Omron Sysmac Studio project Benim_Fonk (Sysmac Studio 1.65.0.64007, StandardProject)

# Controller new_Controller_0: NX1P2-1040DT1 version 1.69
Task PrimaryTask (priority 4, period or condition 2000): Program0

VAR_GLOBAL
    AI_Value2 : REAL;
    OnOff : BOOL;
END_VAR

PROGRAM Program1
VAR
    EnableIn : BOOL;
    EnableOut : BOOL;
    Filtreleme_Start : BOOL;
    Pulse : BOOL;
    Pulse_prev : BOOL;
    Pulse_edge : BOOL;
    Sayici : INT;
    AnalogInput : REAL;
    AnalogArry : ARRAY[1..5] OF REAL;
    Sayici_prev : INT;
    Sayici_chg : BOOL;
    InitDone : BOOL;
    AverageValue : REAL;
END_VAR
(* 
   RUNG 0
   EnableIn -> EnableOut
*)
EnableOut := EnableIn;


(* 
   RUNG 1
   Pulse YÜKSELENKENAR-edge yakala ve Sayici artır
   (Filtreleme_Start TRUE iken)
*)
Pulse_edge := Pulse AND NOT Pulse_prev;
Pulse_prev := Pulse;

IF Filtreleme_Start AND Pulse_edge THEN
    Sayici := Sayici + INT#1;
END_IF;


(* 
   RUNG 2–6 (Optimize)
   Sayici değiştiğinde (Up mantığı gibi tek sefer) ve 1..5 aralığındaysa
   AnalogArry[Sayici] := AnalogInput
 *)
IF NOT InitDone THEN
    Sayici_chg := FALSE;        (* ilk task'ta tetik üretme *)
    Sayici_prev := Sayici;      (* başlangıç referansı *)
    InitDone := TRUE;
ELSE
    Sayici_chg := (Sayici <> Sayici_prev);
    Sayici_prev := Sayici;
END_IF;

IF Sayici_chg AND (Sayici >= INT#1) AND (Sayici <= INT#5) THEN
    AnalogArry[Sayici] := AnalogInput;

    (* 
       RUNG 6 içindeki AryMean
 *)
    IF Sayici = INT#5 THEN
        AverageValue :=
            (AnalogArry[1] + AnalogArry[2] + AnalogArry[3] + AnalogArry[4] + AnalogArry[5]) / REAL#5.0;
    END_IF;
END_IF;


(* 
   RUNG 7
   Sayici > 5 olunca Sayici'yi 1'e çek
   (Ladder'da Up+MOVE var; burada wrap mantığıyla aynı sonucu verir)
 *)
IF Sayici > INT#5 THEN
    Sayici := INT#1;
END_IF;
END_PROGRAM

PROGRAM Program0
VAR
    Scale_Value : REAL;
    Scale_X0 : REAL;
    Scale_Y0 : REAL;
    Scale_X1 : REAL;
    Scale_Y1 : REAL;
    Scale_Out : REAL;
    Lim_Min : REAL;
    Lim_Max : REAL;
    Lim_Out : REAL;
    Analog_Input : REAL;
    InputMin : REAL;
    OutputMin : REAL;
    OutputMax : REAL;
    BasinsDeg : REAL;
    InputMax : REAL;
    BenimFiltre_5liOrt : Filtreleme;
    Ton_Pulse : TON;
    Pulse_200ms : BOOL;
    Ortalama_Deger : REAL;
    OnOff : BOOL;
END_VAR
VAR_EXTERNAL
    AI_Value2 : REAL;
END_VAR
VAR
    _t1 : BOOL;
    _p2 : BOOL;
END_VAR

(* Section Section0: ladder, written here as Structured Text *)

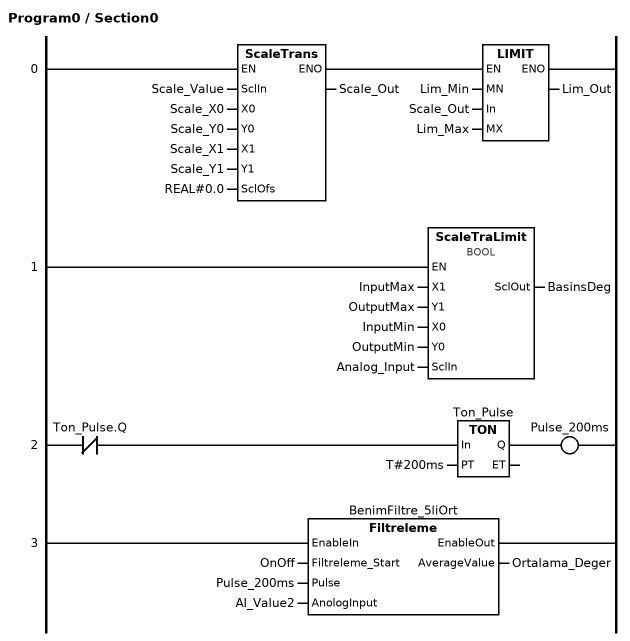
(* Rung 0 *)
Scale_Out := ScaleTrans(SclIn := Scale_Value, X0 := Scale_X0, Y0 := Scale_Y0, X1 := Scale_X1, Y1 := Scale_Y1, SclOfs := REAL#0.0);
Lim_Out := LIMIT(MN := Lim_Min, In := Scale_Out, MX := Lim_Max);
(* Rung 1 *)
_t1 := ScaleTraLimit(X1 := InputMax, Y1 := OutputMax, X0 := InputMin, Y0 := OutputMin, SclIn := Analog_Input, SclOut => BasinsDeg);
(* Rung 2 *)
_p2 := NOT Ton_Pulse.Q;
Ton_Pulse(In := _p2, PT := T#200ms);
Pulse_200ms := Ton_Pulse.Q;
(* Rung 3 *)
BenimFiltre_5liOrt(EnableIn := TRUE, Filtreleme_Start := OnOff, Pulse := Pulse_200ms, AnologInput := AI_Value2, AverageValue => Ortalama_Deger);
END_PROGRAM

FUNCTION ScaleTraLimit : BOOL
VAR
    Scl_Out_Temp : REAL;
END_VAR
VAR_INPUT
    X1 : REAL;
    Y1 : REAL;
    X0 : REAL;
    Y0 : REAL;
    SclIn : REAL;
END_VAR
VAR_OUTPUT
    SclOut : REAL;
END_VAR
(* ladder, written here as Structured Text *)

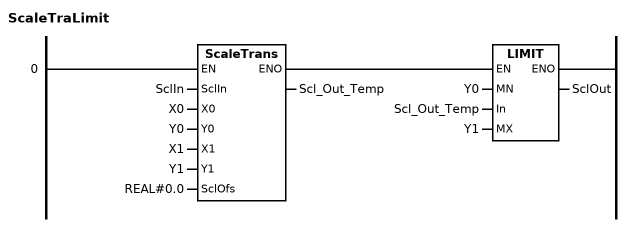
(* Rung 0 *)
Scl_Out_Temp := ScaleTrans(SclIn := SclIn, X0 := X0, Y0 := Y0, X1 := X1, Y1 := Y1, SclOfs := REAL#0.0);
SclOut := LIMIT(MN := Y0, In := Scl_Out_Temp, MX := Y1);
END_FUNCTION

FUNCTION Function0 : BOOL
VAR
    EnableIn : BOOL;
    EnableOut : BOOL;
    Filtreleme_Start : BOOL;
    Pulse : BOOL;
    Pulse_prev : BOOL;
    Pulse_edge : BOOL;
    Sayici : INT;
    AnalogInput : REAL;
    AnalogArry : ARRAY[1..5] OF REAL;
    Sayici_prev : INT;
    Sayici_chg : BOOL;
    InitDone : BOOL;
END_VAR
(* Rung 0 *)
EnableOut := EnableIn;

(* Rung 1 *)
Pulse_edge := Pulse AND NOT Pulse_prev;
Pulse_prev := Pulse;

IF Filtreleme_Start AND Pulse_edge THEN
    Sayici := Sayici + INT#1;
END_IF;

(* Rung 2–6 *)
IF NOT InitDone THEN
    Sayici_chg := FALSE;
    Sayici_prev := Sayici;
    InitDone := TRUE;
ELSE
    Sayici_chg := (Sayici <> Sayici_prev);
    Sayici_prev := Sayici;
END_IF;

IF Sayici_chg AND (Sayici >= INT#1) AND (Sayici <= INT#5) THEN
    AnalogArry[Sayici] := AnalogInput;
END_IF;
END_FUNCTION

FUNCTION_BLOCK Filtreleme
VAR
    Sayici : INT;
    AnologArry : ARRAY[1..5] OF REAL;
END_VAR
VAR_INPUT
    EnableIn : BOOL;
END_VAR
VAR_OUTPUT
    EnableOut : BOOL;
END_VAR
VAR_INPUT
    Filtreleme_Start : BOOL;
    Pulse : BOOL;
    AnologInput : REAL;
END_VAR
VAR_OUTPUT
    AverageValue : REAL;
END_VAR
VAR
    _e1 : R_TRIG;
    _e2 : R_TRIG;
    _e3 : R_TRIG;
    _e4 : R_TRIG;
    _e5 : R_TRIG;
    _e6 : R_TRIG;
    _e7 : R_TRIG;
END_VAR
(* ladder, written here as Structured Text *)

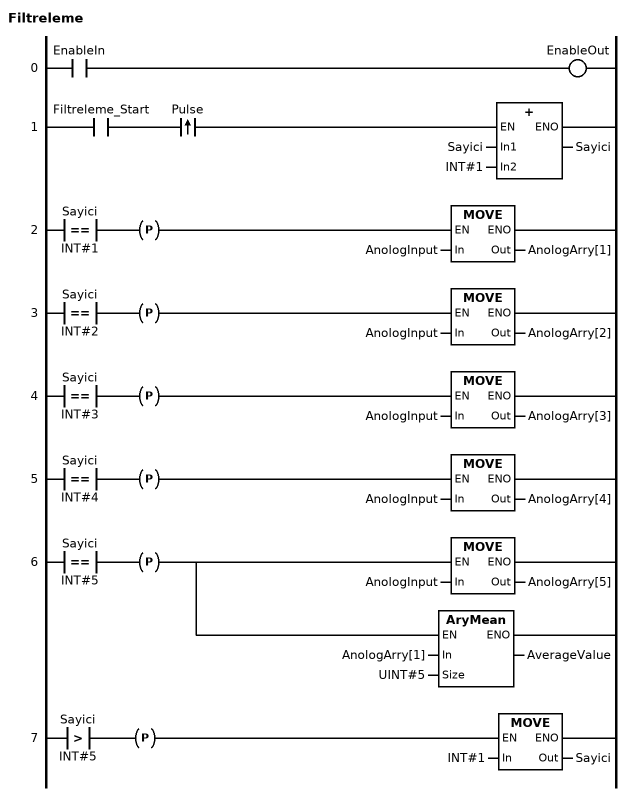
(* Rung 0 *)
EnableOut := EnableIn;
(* Rung 1 *)
_e1(CLK := Pulse);
IF Filtreleme_Start AND _e1.Q THEN Sayici := Sayici + INT#1; END_IF;
(* Rung 2 *)
_e2(CLK := Sayici = INT#1);
IF _e2.Q THEN AnologArry[1] := AnologInput; END_IF;
(* Rung 3 *)
_e3(CLK := Sayici = INT#2);
IF _e3.Q THEN AnologArry[2] := AnologInput; END_IF;
(* Rung 4 *)
_e4(CLK := Sayici = INT#3);
IF _e4.Q THEN AnologArry[3] := AnologInput; END_IF;
(* Rung 5 *)
_e5(CLK := Sayici = INT#4);
IF _e5.Q THEN AnologArry[4] := AnologInput; END_IF;
(* Rung 6 *)
_e6(CLK := Sayici = INT#5);
IF _e6.Q THEN
    AnologArry[5] := AnologInput;
    AverageValue := AryMean(In := AnologArry[1], Size := UINT#5);
END_IF;
(* Rung 7 *)
_e7(CLK := Sayici > INT#5);
IF _e7.Q THEN Sayici := INT#1; END_IF;
END_FUNCTION_BLOCK